// TIA Portal V18 export
TYPE "typeLimitPack"
// stored: IsFailsafeCompliant false
   STRUCT
      x_min : Real;
      x_max : Real;
      y_min : Real;
      y_max : Real;
   END_STRUCT;
END_TYPE
